Staubli VAL3: HIT_YD.dtx

aio aConvSpeed = {link=ModbusSrv-0\Modbus-Word\ao[3]}
aio aPlcCmd = {link=ModbusSrv-0\Modbus-Word\ai[0]}
aio aRbAlarm = {link=ModbusSrv-0\Modbus-Word\ao[0]}
aio aRbStatus = {link=ModbusSrv-0\Modbus-Word\ao[1]}
bool _bConvExist = true
bool _bEndCycle
bool _bIsPicking = true
bool _bIsPlacing
bool _bMutexCnvQueue = true
bool _bPartInTool
bool _bSentToHome
bool bIsPermitPlace = true
bool bIsStartPlace = true
bool bLockPage
bool bPickDetection
bool bSetConvSpeed
bool bSyn
bool bTransferData
dio dAlarm[8]
  [0] = {link=ModbusSrv-0\Modbus-Bit\do[8]}
  [1] = {link=ModbusSrv-0\Modbus-Bit\do[9]}
  [2] = {link=ModbusSrv-0\Modbus-Bit\do[10]}
  [3] = {link=ModbusSrv-0\Modbus-Bit\do[11]}
  [4] = {link=ModbusSrv-0\Modbus-Bit\do[12]}
  [5] = {link=ModbusSrv-0\Modbus-Bit\do[13]}
  [6] = {link=ModbusSrv-0\Modbus-Bit\do[14]}
  [7] = {link=ModbusSrv-0\Modbus-Bit\do[15]}
dio dBlow = {link=BasicIO-1\%Q5}
dio dControlVacuum[4]
  [0] = {link=BasicIO-1\%Q7}
  [1] = {link=BasicIO-1\%Q6}
  [2] = {link=BasicIO-1\%Q5}
  [3] = {link=BasicIO-1\%Q4}
dio dPartInTool = {link=fIn0}
dio dPermitPlace[4]
  [0] = {link=ModbusSrv-0\Modbus-Bit\di[3]}
  [1] = {link=ModbusSrv-0\Modbus-Bit\di[2]}
  [2] = {link=ModbusSrv-0\Modbus-Bit\di[1]}
  [3] = {link=ModbusSrv-0\Modbus-Bit\di[0]}
dio dPlaceDone[4]
  [0] = {link=ModbusSrv-0\Modbus-Bit\do[3]}
  [1] = {link=ModbusSrv-0\Modbus-Bit\do[2]}
  [2] = {link=ModbusSrv-0\Modbus-Bit\do[1]}
  [3] = {link=ModbusSrv-0\Modbus-Bit\do[0]}
dio dStartControl[4]
  [0] = {link=ModbusSrv-0\Modbus-Bit\di[4]}
  [1] = {link=ModbusSrv-0\Modbus-Bit\di[5]}
  [2] = {link=ModbusSrv-0\Modbus-Bit\di[6]}
  [3] = {link=ModbusSrv-0\Modbus-Bit\di[7]}
dio dStartState[4]
  [0] = {link=ModbusSrv-0\Modbus-Bit\do[4]}
  [1] = {link=ModbusSrv-0\Modbus-Bit\do[5]}
  [2] = {link=ModbusSrv-0\Modbus-Bit\do[6]}
  [3] = {link=ModbusSrv-0\Modbus-Bit\do[7]}
dio dVacuum = {link=BasicIO-1\%Q4}
frame fConveyor = {x=690.465999, y=-334.533545, z=-72.519533, rx=0.736674, ry=-0.299775, rz=179.886741, fatherId=world[0]}
frame fDetection = {x=319.933347, y=-456.969728, z=-77.119399, rx=1.134288, ry=-0.307561, rz=179.705392, fatherId=world[0]}
jointRs jDropPart = {j1=-61.262813, j2=45.342289, j3=74.332986, j4=152.342331}
jointRs jHome = {j1=-61.262813, j2=45.342289, j3=74.332986, j4=152.342331}
jointRs jPark = {j1=-61.262813, j2=45.342289, j3=74.332986, j4=152.342331}
mdesc _mLoad = {accel=77.44, vel=88, decel=77.44, leave=30, reach=30}
mdesc mLoad = {accel=121, vel=110, decel=121, leave=30, reach=30}
mdesc mNomSpeed = {accel=144, vel=120, decel=144, leave=20, reach=20}
mdesc mPickDown = {accel=169, vel=130, decel=169, blend=off, leave=30, reach=30}
mdesc mPickup = {accel=144, vel=120, decel=144}
mdesc mPlaceDown = {accel=144, vel=120, decel=144, blend=off, leave=15, reach=15}
mdesc mPlaceUp = {accel=169, vel=130, decel=169, blend=cartesian, leave=20, reach=20}
mdesc mSlow = {accel=1, vel=10, decel=1, leave=10, reach=10}
mdesc mUnload = {accel=144, vel=120, decel=144, leave=40, reach=40}
num _nBlowDelay
num _nCntBypassed
num _nCntPartsDone[2]
  [0] = 59990
  [1] = 59989
num _nCntTransfered = 8399
num _nConvSpd = 557.925928
num _nCycleTime[4]
  [0] = 1.433
  [1] = 0.608
  [2] = 0.75
  [3] = 0.552
num _nCycleTimeIndx = 2
num _nID = 1
num _nLastStateCMD
num _nOmacStat = 3
num _nPartID = 1
num _nPlaceCurItem[2]
num _nPullIndexTQ
num _nPushIndexTQ
num _nStateCMD
num _nTimer = 24802.571
num _nTrackErr = 3106
num nBlowID = 0.5
num nBypass
num nLoadRatio[4]
  [0] = 1.05
  [1] = 0.95
  [2] = 0.8
  [3] = 0.8
num nNomConvSpeed = 100
num nPartHeight = 8
num nPickAppro = 50
num nPickOS_X = -3
num nPickOS_Y
num nPlaceAppro = 50
num nPlaceCycleNum = 3
public num nPlaceNum = 3
num nSafeMaxX = 850
num nSafeMaxY = 850
num nSafeMinX = -850
num nSafeMinY = -850
num nTestData[5]
  [0] = 2
  [1] = -49
  [2] = 51
  [3] = 1
  [4] = 10107
num nVacuumID = 0.2
num nWaitDist2Up4BP = -150
num nWaitDistToDown = 50
num nWaitDistToUp[1 3]
  [0,0] = -80
  [0,1] = 150
  [0,2] = 400
num nWaitDistX = -150
object _oTransferQueue[1 100]
  [0,0]
    num nID = -1
    num nLatchedValue
    trsf trTrsf
  [0,1]
    num nID = -1
    num nLatchedValue
    trsf trTrsf
  [0,2]
    num nID = -1
    num nLatchedValue
    trsf trTrsf
  [0,3]
    num nID = -1
    num nLatchedValue
    trsf trTrsf
  [0,4]
    num nID = -1
    num nLatchedValue
    trsf trTrsf
  [0,5]
    num nID = -1
    num nLatchedValue
    trsf trTrsf
  [0,6]
    num nID = -1
    num nLatchedValue
    trsf trTrsf
  [0,7]
    num nID = -1
    num nLatchedValue
    trsf trTrsf
  [0,8]
    num nID = -1
    num nLatchedValue
    trsf trTrsf
  [0,9]
    num nID = -1
    num nLatchedValue
    trsf trTrsf
  [0,10]
    num nID = -1
    num nLatchedValue
    trsf trTrsf
  [0,11]
    num nID = -1
    num nLatchedValue
    trsf trTrsf
  [0,12]
    num nID = -1
    num nLatchedValue
    trsf trTrsf
  [0,13]
    num nID = -1
    num nLatchedValue
    trsf trTrsf
  [0,14]
    num nID = -1
    num nLatchedValue
    trsf trTrsf
  [0,15]
    num nID = -1
    num nLatchedValue
    trsf trTrsf
  [0,16]
    num nID = -1
    num nLatchedValue
    trsf trTrsf
  [0,17]
    num nID = -1
    num nLatchedValue
    trsf trTrsf
  [0,18]
    num nID = -1
    num nLatchedValue
    trsf trTrsf
  [0,19]
    num nID = -1
    num nLatchedValue
    trsf trTrsf
  [0,20]
    num nID = -1
    num nLatchedValue
    trsf trTrsf
  [0,21]
    num nID = -1
    num nLatchedValue
    trsf trTrsf
  [0,22]
    num nID = -1
    num nLatchedValue
    trsf trTrsf
  [0,23]
    num nID = -1
    num nLatchedValue
    trsf trTrsf
  [0,24]
    num nID = -1
    num nLatchedValue
    trsf trTrsf
  [0,25]
    num nID = -1
    num nLatchedValue
    trsf trTrsf
  [0,26]
    num nID = -1
    num nLatchedValue
    trsf trTrsf
  [0,27]
    num nID = -1
    num nLatchedValue
    trsf trTrsf
  [0,28]
    num nID = -1
    num nLatchedValue
    trsf trTrsf
  [0,29]
    num nID = -1
    num nLatchedValue
    trsf trTrsf
  [0,30]
    num nID = -1
    num nLatchedValue
    trsf trTrsf
  [0,31]
    num nID = -1
    num nLatchedValue
    trsf trTrsf
  [0,32]
    num nID = -1
    num nLatchedValue
    trsf trTrsf
  [0,33]
    num nID = -1
    num nLatchedValue
    trsf trTrsf
  [0,34]
    num nID = -1
    num nLatchedValue
    trsf trTrsf
  [0,35]
    num nID = -1
    num nLatchedValue
    trsf trTrsf
  [0,36]
    num nID = -1
    num nLatchedValue
    trsf trTrsf
  [0,37]
    num nID = -1
    num nLatchedValue
    trsf trTrsf
  [0,38]
    num nID = -1
    num nLatchedValue
    trsf trTrsf
  [0,39]
    num nID = -1
    num nLatchedValue
    trsf trTrsf
  [0,40]
    num nID = -1
    num nLatchedValue
    trsf trTrsf
  [0,41]
    num nID = -1
    num nLatchedValue
    trsf trTrsf
  [0,42]
    num nID = -1
    num nLatchedValue
    trsf trTrsf
  [0,43]
    num nID = -1
    num nLatchedValue
    trsf trTrsf
  [0,44]
    num nID = -1
    num nLatchedValue
    trsf trTrsf
  [0,45]
    num nID = -1
    num nLatchedValue
    trsf trTrsf
  [0,46]
    num nID = -1
    num nLatchedValue
    trsf trTrsf
  [0,47]
    num nID = -1
    num nLatchedValue
    trsf trTrsf
  [0,48]
    num nID = -1
    num nLatchedValue
    trsf trTrsf
  [0,49]
    num nID = -1
    num nLatchedValue
    trsf trTrsf
  [0,50]
    num nID = -1
    num nLatchedValue
    trsf trTrsf
  [0,51]
    num nID = -1
    num nLatchedValue
    trsf trTrsf
  [0,52]
    num nID = -1
    num nLatchedValue
    trsf trTrsf
  [0,53]
    num nID = -1
    num nLatchedValue
    trsf trTrsf
  [0,54]
    num nID = -1
    num nLatchedValue
    trsf trTrsf
  [0,55]
    num nID = -1
    num nLatchedValue
    trsf trTrsf
  [0,56]
    num nID = -1
    num nLatchedValue
    trsf trTrsf
  [0,57]
    num nID = -1
    num nLatchedValue
    trsf trTrsf
  [0,58]
    num nID = -1
    num nLatchedValue
    trsf trTrsf
  [0,59]
    num nID = -1
    num nLatchedValue
    trsf trTrsf
  [0,60]
    num nID = -1
    num nLatchedValue
    trsf trTrsf
  [0,61]
    num nID = -1
    num nLatchedValue
    trsf trTrsf
  [0,62]
    num nID = -1
    num nLatchedValue
    trsf trTrsf
  [0,63]
    num nID = -1
    num nLatchedValue
    trsf trTrsf
  [0,64]
    num nID = -1
    num nLatchedValue
    trsf trTrsf
  [0,65]
    num nID = -1
    num nLatchedValue
    trsf trTrsf
  [0,66]
    num nID = -1
    num nLatchedValue
    trsf trTrsf
  [0,67]
    num nID = -1
    num nLatchedValue
    trsf trTrsf
  [0,68]
    num nID = -1
    num nLatchedValue
    trsf trTrsf
  [0,69]
    num nID = -1
    num nLatchedValue
    trsf trTrsf
  [0,70]
    num nID = -1
    num nLatchedValue
    trsf trTrsf
  [0,71]
    num nID = -1
    num nLatchedValue
    trsf trTrsf
  [0,72]
    num nID = -1
    num nLatchedValue
    trsf trTrsf
  [0,73]
    num nID = -1
    num nLatchedValue
    trsf trTrsf
  [0,74]
    num nID = -1
    num nLatchedValue
    trsf trTrsf
  [0,75]
    num nID = -1
    num nLatchedValue
    trsf trTrsf
  [0,76]
    num nID = -1
    num nLatchedValue
    trsf trTrsf
  [0,77]
    num nID = -1
    num nLatchedValue
    trsf trTrsf
  [0,78]
    num nID = -1
    num nLatchedValue
    trsf trTrsf
  [0,79]
    num nID = -1
    num nLatchedValue
    trsf trTrsf
  [0,80]
    num nID = -1
    num nLatchedValue
    trsf trTrsf
  [0,81]
    num nID = -1
    num nLatchedValue
    trsf trTrsf
  [0,82]
    num nID = -1
    num nLatchedValue
    trsf trTrsf
  [0,83]
    num nID = -1
    num nLatchedValue
    trsf trTrsf
  [0,84]
    num nID = -1
    num nLatchedValue
    trsf trTrsf
  [0,85]
    num nID = -1
    num nLatchedValue
    trsf trTrsf
  [0,86]
    num nID = -1
    num nLatchedValue
    trsf trTrsf
  [0,87]
    num nID = -1
    num nLatchedValue
    trsf trTrsf
  [0,88]
    num nID = -1
    num nLatchedValue
    trsf trTrsf
  [0,89]
    num nID = -1
    num nLatchedValue
    trsf trTrsf
  [0,90]
    num nID = -1
    num nLatchedValue
    trsf trTrsf
  [0,91]
    num nID = -1
    num nLatchedValue
    trsf trTrsf
  [0,92]
    num nID = -1
    num nLatchedValue
    trsf trTrsf
  [0,93]
    num nID = -1
    num nLatchedValue
    trsf trTrsf
  [0,94]
    num nID = -1
    num nLatchedValue
    trsf trTrsf
  [0,95]
    num nID = -1
    num nLatchedValue
    trsf trTrsf
  [0,96]
    num nID = -1
    num nLatchedValue
    trsf trTrsf
  [0,97]
    num nID = -1
    num nLatchedValue
    trsf trTrsf
  [0,98]
    num nID = -1
    num nLatchedValue
    trsf trTrsf
  [0,99]
    num nID = -1
    num nLatchedValue
    trsf trTrsf
pointRs pPick = {x=-54, y=-28, rz=72.6, shoulder=righty, fatherId=fDetection[0]}
pointRs pPlace[4]
  [0] = {x=752.590073, y=-120.83, z=-69.15, rx=180, rz=90.41, shoulder=righty, fatherId=world[0]}
  [1] = {x=614.985623, y=-120.83, z=-69.15, rx=180, rz=90.41, shoulder=righty, fatherId=world[0]}
  [2] = {x=479.250185, y=-120.83, z=-69.15, rx=180, rz=90.41, shoulder=righty, fatherId=world[0]}
  [3] = {x=345.150595, y=-120.83, z=-69.15, rx=180, rz=90.41, shoulder=righty, fatherId=world[0]}
sio sClient = {link=Socket\synRobot2}
sio skToRobot = {link=Socket\toRobot_sk1}
string _sCycleStatus = "Distance to pick:  -70.37"
string sConveyorList = "cvIn"
string sSecondRStatus
string sString = "done"
tool tGripper = {z=75, rz=-128, fatherId=flange[0], ioLink=valve1}
public trsf trTrsfPlace[4]
  [1] = {x=140}
  [2] = {x=280}
  [3] = {x=420}
